(* IEC 61131-3 sources: RAG_PLC/data/result/test/044, 2 files *)

(* ---- wrapped.st ---- *)
(* =========================================================
   Generated by PLC-Eval Benchmark Wrapper
   ========================================================= *)

FUNCTION_BLOCK LLM_Wrapper_FB
VAR_INPUT
    IN : oscat_STRING250;
    CX : STRING;
END_VAR

VAR_OUTPUT
    DEL_CHARS : oscat_STRING250;
END_VAR

VAR
    pos : INT;
    stop : INT;
    char : oscat_STRING1;
END_VAR

DEL_CHARS := IN;
stop := LEN(IN);
pos := 1;
WHILE pos <= stop DO
    char := MID(DEL_CHARS, pos, 1);
    IF FIND(CX, char) > 0 THEN
        DEL_CHARS := DELETE(DEL_CHARS, pos, 1);
        stop := stop - 1; (* 现在字符串长度减一 *)
    ELSE
        pos := pos + 1; (* 字符未找到，跳到下一个 *)
    END_IF;
END_WHILE;
END_FUNCTION_BLOCK

PROGRAM Auto_Proxy_Prg
  VAR
    instance : LLM_Wrapper_FB;
  END_VAR

  instance();
END_PROGRAM

CONFIGURATION Config0
  RESOURCE Res0 ON PLC
    TASK TaskMain(INTERVAL := T#20ms, PRIORITY := 0);
    PROGRAM Inst0 WITH TaskMain : Auto_Proxy_Prg;
  END_RESOURCE
END_CONFIGURATION

(* ---- raw_code.st ---- *)
VAR_INPUT
    IN : oscat_STRING250;
    CX : STRING;
END_VAR

VAR_OUTPUT
    DEL_CHARS : oscat_STRING250;
END_VAR

VAR
    pos : INT;
    stop : INT;
    char : oscat_STRING1;
END_VAR

DEL_CHARS := IN;
stop := LEN(IN);
pos := 1;
WHILE pos <= stop DO
    char := MID(DEL_CHARS, pos, 1);
    IF FIND(CX, char) > 0 THEN
        DEL_CHARS := DELETE(DEL_CHARS, pos, 1);
        stop := stop - 1; (* 现在字符串长度减一 *)
    ELSE
        pos := pos + 1; (* 字符未找到，跳到下一个 *)
    END_IF;
END_WHILE;
